PROGRAM EM05_Counters
VAR
	ref_Master: REFERENCE TO UDT_AXISADMIN;
	Ref_MachineStateModel: REFERENCE TO PackMlv3_StateModel;
	Ref_Unit: REFERENCE TO UDT_UnitAdmin;	
	
	ref_Work_Recipe: REFERENCE TO UDT_Hmi_Output; //当前生产的配方反馈给触摸屏
	ref_diBeltObjCnt: REFERENCE TO DINT;
	ref_lrLatchMasterPos: REFERENCE TO LREAL;
    ref_lrMasterTargetPos: REFERENCE TO LREAL;
	ref_BinList: REFERENCE TO UDT_BINlist;
	
	EM_No: INT:=5;
	diProductCnt: DINT;
	tonAbortingWatchDog: TON;
	i,j,k: INT;

	rt_ProductCntUp: R_Trig;
	
	arDropFlag: ARRAY[1..40] OF BOOL;//落料标志	
	arDropCnt: ARRAY[1..40] OF DINT;//落料技数


	tonExeRtirg: ARRAY [1..40 ] OF Ton;
	arDropInRange: ARRAY [1..40 ] OF BOOL;
	d: INT;
	rtDropInRange: ARRAY [1..40 ] OF R_trig;
	ftDropFlag: ARRAY [1..40 ] OF F_trig;
	rtDropFlag: ARRAY [1..40 ] OF R_trig;
	ftInSensor: ARRAY [1..40 ] OF F_trig;
	rtInSensor: ARRAY [1..40 ] OF R_trig;
	ftOutSensor: ARRAY [1..40 ] OF F_trig;
	rtOutSensor: ARRAY [1..40 ] OF R_trig;	

	iNotDone: INT;

	iHomeCnt: INT;
	iPowerCnt: INT;
	iInitDone: INT;
	iStandstill: INT;
	Loc_Counter_Seq: INT;

	diMasterRangeCnt: DINT; //出料皮带计数
	aoi_binProduct: AOI_BIN;
	rtBeltInRange: R_trig;
	lrMasterPosAdd: LREAL;
	lrWorkPosBuffer: LREAL;
	iNotInitID: INT;

	iMovAbsCnt: INT;

	lrWorkPosExe: LREAL;
	iC: INT;
	iB: INT;
	iMovFailCnt: INT;
	
	
	tonCounterSeq: Ton;
	CounterSeq: SequenceTransfer;
	
	iDrop: INT;
	iBusyCounter: INT;
	iNotBusyCounter: INT;
	iCntDone: INT;
END_VAR

VAR CONSTANT
;
END_VAR

//伺服转1圈 落料24颗
Ref_MachineStateModel REF= UN01_MachineStateModel;
Ref_Unit REF=Unit01;
ref_Work_Recipe REF=HMI_Output;
ref_Master REF= arVirtualAxisAdmin[1];
ref_diBeltObjCnt REF=glb_diBeltObjCnt;

ref_BinList REF= Glb_BinList;
MainRoution();

ACTION CM01_Counters:
CASE CounterSeq.Now OF
	0: 
	   IF Ref_MachineStateModel.Sts_Resetting THEN
          CounterSeq(ExeCute:= TRUE, Next:= Seq_Resetting);
	   END_IF	
	   IF Ref_MachineStateModel.Sts_Stopping  THEN
          CounterSeq(ExeCute:= TRUE, Next:= Seq_Stopping);
	   END_IF
	   IF Ref_MachineStateModel.Sts_Execute  THEN
		  CounterSeq(ExeCute:= TRUE, Next:= 110);   
	   END_IF	 	   
	Seq_Resetting:
	  iPowerCnt:=0;
		FOR i:=1 TO 40 DO
			IF NOT arRealAxisAdmin[i].o.PowerOn THEN
			   arRealAxisAdmin[i].i.Enable:=TRUE;
			ELSE
			   iPowerCnt:=iPowerCnt+1;
			END_IF  
		END_FOR
		IF iPowerCnt=40 THEN
		   CounterSeq(ExeCute:= TRUE, Next:= 11);
		END_IF
		IF Ref_MachineStateModel.Sts_Stopping  THEN
		   CounterSeq(ExeCute:= TRUE, Next:= Seq_Stopping);
		END_IF	  
		
	11:
       tonCounterSeq(IN:=TRUE , PT:=T#1S , Q=> , ET=> );
	   IF tonCounterSeq.Q THEN
          tonCounterSeq(IN:=FALSE , PT:=T#1S , Q=> , ET=> );	
          CounterSeq(ExeCute:= TRUE, Next:= 20);
	   END_IF
	   
	20:
		IF NOT glb_AllAxisHomed_UN01 THEN
			CounterSeq(ExeCute:=TRUE , Next:= 21);  
			ELSE
			CounterSeq(ExeCute:=TRUE , Next:= 30); 
		END_IF	
	21:
	   iHomeCnt:=0;
	   FOR i:=1 TO 40 DO
		   arRealAxisAdmin[i].i.Pos:=0;
		   arRealAxisAdmin[i].i.HomeMode:=2;
		   arRealAxisAdmin[i].i.Home:=TRUE;    
		   IF arRealAxisAdmin[i].o.HomeDone THEN
			   iHomeCnt:=iHomeCnt+1;
		   END_IF     
	   END_FOR   
	   
	   IF iHomeCnt=40 THEN
          CounterSeq(ExeCute:= TRUE, Next:= 22);
	   END_IF	
       IF Ref_MachineStateModel.Sts_Stopping  THEN
	      CounterSeq(ExeCute:= TRUE, Next:= Seq_Stopping);
	   END_IF
		   
    22:
       tonCounterSeq(IN:=TRUE , PT:=T#1S , Q=> , ET=> );
	   IF tonCounterSeq.Q THEN
          tonCounterSeq(IN:=FALSE , PT:=T#1S , Q=> , ET=> );	
          CounterSeq(ExeCute:= TRUE, Next:= 23);
	   END_IF
          
	23:
       FOR  i:=1 TO 40 DO
		   arRealAxisAdmin[i].i.Home:=FALSE;
	   END_FOR

       CounterSeq(ExeCute:= TRUE, Next:= 30);
   
	30:
	    iNotBusyCounter:=0;
	    FOR i:=1 TO 40 DO
			IF NOT arCounters[i].Busy THEN
				iNotBusyCounter:=iNotBusyCounter+1;
			ELSE
				iBusyCounter:=i;
			END_IF	
		END_FOR
		IF iNotBusyCounter=40 THEN
           CounterSeq(ExeCute:= TRUE, Next:= 40);
	    ELSE IF Ref_MachineStateModel.Sts_Stopping  THEN
			    CounterSeq(ExeCute:= TRUE, Next:= Seq_Stopping);
			 END_IF	
		END_IF
		
    40:		
		tonCounterSeq(IN:=TRUE , PT:=T#1S , Q=> , ET=> );
		IF tonCounterSeq.Q THEN
		   tonCounterSeq(IN:=FALSE , PT:=T#1S , Q=> , ET=> );	
		   CounterSeq(ExeCute:= TRUE, Next:= Seq_ResettingDone);
		END_IF    

	Seq_ResettingDone:
		IF NOT Ref_MachineStateModel.Sts_Resetting THEN
		   CounterSeq(ExeCute:= TRUE, Next:= 0);
		END_IF	
	  
    110:
		   IF HMI_Output.RecipeModifyDone THEN
				FOR i:=1 TO 40 DO 
					arCounters[i].Enable:=TRUE;		
				END_FOR	
           ELSE
				FOR i:=1 TO 40 DO 
					arCounters[i].Enable:=FALSE;		
				END_FOR				   
		   END_IF
	
		
	   IF Ref_MachineStateModel.Sts_Stopping  THEN
          CounterSeq(ExeCute:= TRUE, Next:= Seq_Stopping);
	   END_IF		
		
		
		
		
	Seq_Stopping: 	
		iNotBusyCounter:=0;
		FOR i:=1 TO 40 DO
			IF NOT arCounters[i].Busy THEN
				iNotBusyCounter:=iNotBusyCounter+1;
			ELSE
				iBusyCounter:=i;
			END_IF	
		END_FOR
		IF iNotBusyCounter=40 THEN
		   CounterSeq(ExeCute:= TRUE, Next:= 903);
		END_IF
	
	
	903:
		FOR i:=1 TO 40 DO 
			arCounters[i].Enable:=FALSE;	
            arCounters[i].Execute:=FALSE;	
            CounterSeq(ExeCute:= TRUE, Next:= 904);	
		END_FOR	
    904:
		tonCounterSeq(IN:=TRUE , PT:=T#1.5S , Q=> , ET=> );	  
		IF tonCounterSeq.Q THEN
			tonCounterSeq(IN:=FALSE , PT:=T#1.5S , Q=> , ET=> );	
			CounterSeq(ExeCute:= TRUE, Next:= 905);  
		END_IF				

	905:
	    FOR i:=1 TO 40 DO 
			arRealAxisAdmin[i].i.Disable:=TRUE;
			CounterSeq(ExeCute:= TRUE, Next:= Seq_StoppingDone);
        END_FOR	
			
	
	Seq_StoppingDone:
		IF NOT Ref_MachineStateModel.Sts_Stopping THEN
		   CounterSeq(ExeCute:= TRUE, Next:= 0);
		END_IF	
		
END_CASE
END_ACTION

ACTION MainRoution:
EM_No:=5;
IF Ref_Unit.EM_Selected[EM_No] THEN
	IF Ref_MachineStateModel.Sts_Holding THEN
		Ref_Unit.EM_Holding_Done[EM_No]:=TRUE;
		ELSE
		Ref_Unit.EM_Holding_Done[EM_No]:=FALSE;
	END_IF
	IF Ref_MachineStateModel.Sts_UnHolding THEN
		Ref_Unit.EM_UnHolding_Done[EM_No]:=TRUE;
		ELSE
		Ref_Unit.EM_UnHolding_Done[EM_No]:=FALSE;
	END_IF
	
	IF Ref_MachineStateModel.Sts_Suspending THEN
		Ref_Unit.EM_Suspending_Done[EM_No]:=TRUE;
		ELSE
		Ref_Unit.EM_Suspending_Done[EM_No]:=FALSE;
	END_IF
	
	IF Ref_MachineStateModel.Sts_UnSuspending THEN
		Ref_Unit.EM_UnSuspending_Done[EM_No]:=TRUE;
		ELSE
		Ref_Unit.EM_UnSuspending_Done[EM_No]:=FALSE;
	END_IF
	
	IF Ref_MachineStateModel.Sts_Resetting AND CounterSeq.Now=Seq_ResettingDone THEN
       Ref_Unit.EM_Resetting_Done[EM_No]:=TRUE;
       ELSE   
       Ref_Unit.EM_Resetting_Done[EM_No]:=FALSE;	   
	END_IF
	
	IF Ref_MachineStateModel.Sts_Clearing THEN
	   Ref_Unit.EM_Clearing_Done[EM_No]:=TRUE;
	   ELSE   
	   Ref_Unit.EM_Clearing_Done[EM_No]:=FALSE;
	END_IF
	
	IF Ref_MachineStateModel.Sts_Starting THEN
	   Ref_Unit.EM_Starting_Done[EM_No]:=TRUE;
	   ELSE	   
	   Ref_Unit.EM_Starting_Done[EM_No]:=FALSE;
	END_IF
	
	IF Ref_MachineStateModel.Sts_Stopping AND CounterSeq.Now=Seq_StoppingDone THEN
	   Ref_Unit.EM_Stopping_Done[EM_No]:=TRUE;	
	   ELSE
	   Ref_Unit.EM_Stopping_Done[EM_No]:=FALSE;	   
	END_IF

	IF Ref_MachineStateModel.Sts_Aborting THEN
		CounterSeq(ExeCute:= TRUE, Next:= 0);
        FOR i:=1 TO 40 DO 
			arCounters[i].Enable:=FALSE; 
			arDropCylinder[i].i.ActiveIn:=FALSE;
			arDropCylinder[i].i.ActiveOut:=FALSE;
		END_FOR
		
		IF  tonAbortingWatchDog.Q THEN 
		    Ref_Unit.EM_Aborting_Done[EM_No]:=TRUE;
			FOR i:=1 TO 40 DO 
				arRealAxisAdmin[i].i.Enable:=FALSE;
			END_FOR			
		END_IF
		ELSE
        Ref_Unit.EM_Aborting_Done[EM_No]:=FALSE;
	END_IF
	tonAbortingWatchDog(IN:= Ref_MachineStateModel.Sts_Aborting, PT:=T#3S , Q=> , ET=> );	
CM01_Counters();
ELSE
	CounterSeq(ExeCute:= TRUE, Next:= 0);
END_IF
END_ACTION

ACTION SR999_FaultHandler:
;
END_ACTION

END_PROGRAM

(* stored: Version 1.1.0.1, ProductVersion 3.1.4022.16
   POU EM05_Counters: Id {0baf6a8a-1073-4fd6-8135-58eda79fb4c3}, SpecialFunc None
   Action CM01_Counters: Id {88a9805c-ef01-4f14-bfb7-655ee7439444}
   Action MainRoution: Id {7ac38113-d258-4703-b30c-25bd358c8261}
   Action SR999_FaultHandler: Id {f318dec9-3e3e-41d2-af56-7df73e16b5cb} *)
